{attribute 'qualified_only'}
VAR_GLOBAL
		stAxis_1 : AXIS_REF;
		stAxis_2 : AXIS_REF;
		stAxis_3 : AXIS_REF;
		stAxis_4 : AXIS_REF;
END_VAR

(* stored: Version 1.1.0.1, ProductVersion 3.1.4024.0
   GVL GVL: Id {ae16aa83-5e48-4609-bd62-bae9f5908323} *)
